{attribute 'linkalways'} 
{attribute 'no_explicit_call' := 'This FB is a CLASS and must be accessed using methods or properties'}
{attribute 'enable_dynamic_creation'}
FUNCTION_BLOCK FINAL GT_LREAL EXTENDS Node
VAR
	in1 : _LREAL(0.0);
	in2 : _LREAL(0.0);
	out : _BOOL(FALSE);
END_VAR

METHOD PUBLIC Clone : I_Node
VAR
	pNode : POINTER TO GT_LREAL;
END_VAR
pNode := __NEW(GT_LREAL);
Clone := pNode^;
END_METHOD

METHOD FB_init : BOOL
VAR_INPUT
	bInitRetains : BOOL; // if TRUE, the retain variables are initialized (warm start / cold start)
	bInCopyCode : BOOL;  // if TRUE, the instance afterwards gets moved into the copy code (online change)
END_VAR
AddInput('in1',THIS^.in1);
AddInput('in2',THIS^.in2);
AddOutput('out', THIS^.out);
END_METHOD

METHOD PROTECTED OnExecute
VAR
END_VAR
out.Value := in1.Value > in2.Value;
END_METHOD

END_FUNCTION_BLOCK

(* stored: Version 1.1.0.1, ProductVersion 3.1.4024.15
   POU GT_LREAL: Id {72852240-f432-4fb1-8c0b-58ac8e2068b8}, SpecialFunc None
   Folder Constructor: Id {65855179-4819-416f-93da-b7c60886c6c7}
   Method Clone: Id {f393411a-cdb3-44a4-985d-700095d513e9}
   Method FB_init: Id {2bc0c330-8b1a-4016-8525-4d3cf0611f05}
   Method OnExecute: Id {c6b4dd2a-73a2-436c-8525-4c49604c4500} *)
